(* PLC project RefrigeratorControl.project, CODESYS CODESYS V3.5 SP21 Patch 1 *)
(* stored: creationDateTime 2025-11-12T17:51:44.3164415, modificationDateTime 2025-11-12T17:46:05.0958991 *)

(* The program activates or deactivates the cooling compressor depending on the deviaton of the actual temperature from the septpoint temperature (with a hysteresis) TRUE or FALSE of the cooling compresseor is transfered to the signal processing. *)
PROGRAM PLC_PRG
  VAR
    SR_0 : SR;
    Hysteresis : REAL := 1.0;
  END_VAR
  VAR  (* added by the conversion: wires and edge detectors of the diagram *)
    _ADD7_OUT : ANY;
    _LT13_OUT : BOOL;
  END_VAR

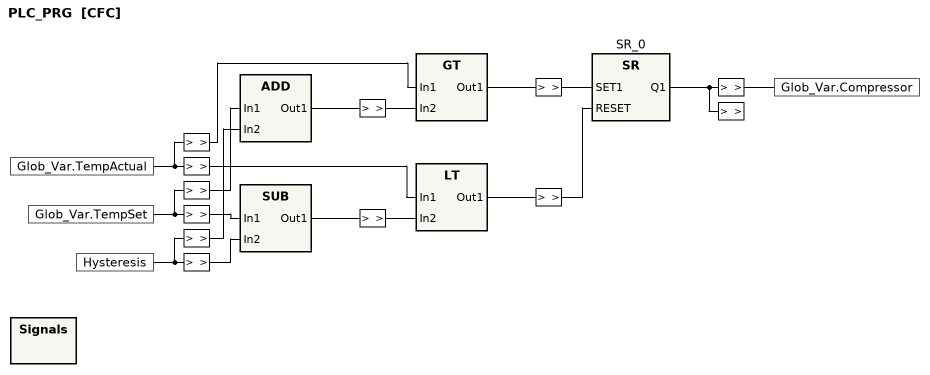
(* CFC diagram, written out as Structured Text *)
Glob_Var.Compressor := SR_0.Q1;
SR_0(SET1 := Glob_Var.TempActual > _ADD7_OUT, RESET := _LT13_OUT);
_ADD7_OUT := Glob_Var.TempSet + Hysteresis;
_LT13_OUT := Glob_Var.TempActual < Glob_Var.TempSet - Hysteresis;
Signals();
END_PROGRAM

PROGRAM Signals
  VAR
    TON_0 : TON;
    TON_1 : TON;
    tSignalTime : TIME := TIME#1s0ms;
    BLINK_0 : BLINK;
  END_VAR

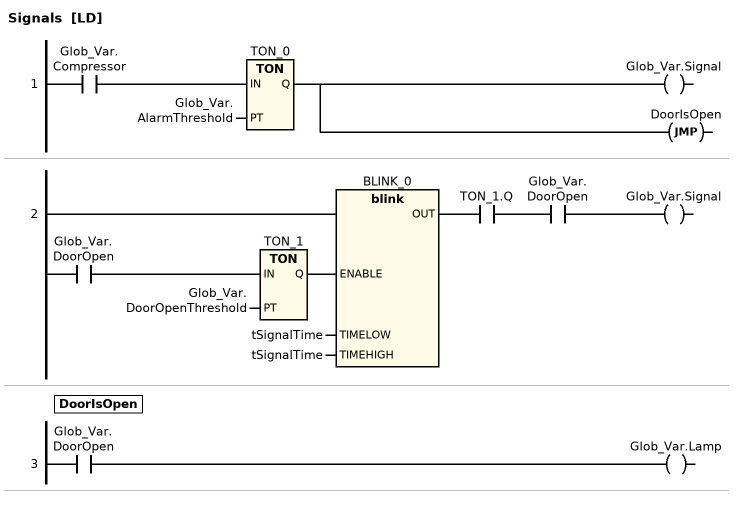
(* LD diagram, written out as Structured Text *)

TON_0(IN := Glob_Var.Compressor, PT := Glob_Var.AlarmThreshold);
Glob_Var.Signal := TON_0.Q;
IF TON_0.Q THEN JMP DoorIsOpen; END_IF;

TON_1(IN := Glob_Var.DoorOpen, PT := Glob_Var.DoorOpenThreshold);
BLINK_0(ENABLE := TON_1.Q, TIMELOW := tSignalTime, TIMEHIGH := tSignalTime);
Glob_Var.Signal := BLINK_0.OUT AND TON_1.Q AND Glob_Var.DoorOpen;
DoorIsOpen:

Glob_Var.Lamp := Glob_Var.DoorOpen;
END_PROGRAM

PROGRAM Simulation
  VAR
    T1 : TON;  (* The temperature is decreased on a time delay, when the comepressor has been activated *)
    P_Cooling : TIME := TIME#500ms;
    xReduceTemp : BOOL;  (* Signal for dereasing the temperature *)
    T2 : TON;  (* The temperature is increased on a time delay, when the compressor has been activated *)
    P_Environment : TIME := TIME#2s0ms;  (* Delay time when the door is closed *)
    P_EnvironmentDoorOpen : TIME := TIME#1s0ms;  (* Delay time when the door is open *)
    xRaiseTemp : BOOL;  (* Signal for increasing the temperature *)
    tTemp : TIME;  (* Delay time *)
  END_VAR

                    // After the compressor has been activated due to TempActual being too high, the temperature decreases.
// The temperature is decremented by 0.1°C per cycle after a delay of P_Cooling
IF Glob_Var.Compressor THEN
	T1(IN:= Glob_Var.Compressor, PT:= P_Cooling, Q=>xReduceTemp);
	IF xReduceTemp THEN
		Glob_Var.TempActual := Glob_Var.TempActual-0.1;
		T1(IN:=FALSE);
	END_IF
END_IF

//If the door is open, the warming occurs faster; SEL selects P_EnvironmentDoorOpen
tTemp:=SEL(Glob_Var.DoorOpen, P_Environment, P_EnvironmentDoorOpen);

//If the compressor is not in operation, then the cooling chamber becomes warmer.
//The  temperature is incremented by 0.1°C per cycle after a delay of tTemp
T2(IN:= TRUE, PT:= tTemp, Q=>xRaiseTemp);	
IF xRaiseTemp THEN
	Glob_Var.TempActual := Glob_Var.TempActual + 0.1;
	T2(IN:=FALSE);
END_IF

                  
END_PROGRAM

CONFIGURATION Device
  RESOURCE Application ON PLC
    {attribute 'qualified_only'}
    VAR_GLOBAL  (* Glob_Var *)
      TempActual : REAL := 8.0;  (* Inputs *)
      TempSet : REAL := 8.0;
      DoorOpen : BOOL;
      AlarmThreshold : TIME := TIME#10s0ms;
      DoorOpenThreshold : TIME := TIME#10s0ms;
      Compressor : BOOL;  (* Outputs *)
      Signal : BOOL;
      Lamp : BOOL;
    END_VAR
    TASK MainTask(INTERVAL := T#20ms, PRIORITY := 1);
    TASK VISU_TASK(INTERVAL := T#100ms, PRIORITY := 31);
    PROGRAM PLC_PRG WITH MainTask : PLC_PRG;
    PROGRAM Simulation WITH MainTask : Simulation;
    PROGRAM VisuElems.Visu_Prg WITH VISU_TASK : VisuElems.Visu_Prg;
  END_RESOURCE
END_CONFIGURATION
